// TIA Portal V16 export
// export: Created 2021-06-25T07:14:34.9561017Z, ExportSetting WithDefaults, DisplayName Totally Integrated Automation Portal, DisplayVersion V16, DisplayName TIA Portal Version Control Interface, DisplayVersion V16, DisplayName TIA Portal Openness, DisplayVersion V16, DisplayName STEP 7 Professional, DisplayVersion V16, DisplayName STEP 7 Safety, DisplayVersion V16, DisplayName WinCC Advanced, DisplayVersion V16
TYPE "udtTest"
// stored: IsFailsafeCompliant false
   STRUCT
      Input : Struct
         signal : Bool;
         block : Bool;
      END_STRUCT;
      Output : Struct
         value : Bool;
         Error : Bool;
      END_STRUCT;
   END_STRUCT;
END_TYPE
